# EPICS autosave request: iocs/pvcamIOC/iocBoot/iocPvCam/auto_settings.req
file "pvCam_settings.req",  	    P=$(P),  R=cam1:
file "NDStdArrays_settings.req",  P=$(P),  R=image:
file "commonPlugin_settings.req", P=$(P)
